// TIA Portal V17 export
// export: Created 2023-04-03T06:31:28.5466402Z, ExportSetting WithDefaults, DisplayName Totally Integrated Automation Portal, DisplayVersion V17 Update 4, DisplayName TIA Portal Openness, DisplayVersion V17 Update 4, DisplayName TIA Portal Version Control Interface, DisplayVersion V17, DisplayName STEP 7 Professional, DisplayVersion V17 Update 4, DisplayName STEP 7 Safety, DisplayVersion V17, DisplayName WinCC Professional, DisplayVersion V17 Update 4
DATA_BLOCK "PCS_2"   // DB43
{ S7_Optimized_Access := 'TRUE' }
VERSION : 0.1
// stored: AutoNumber true, DBAccessibleFromOPCUA true, DBAccessibleFromWebserver true, IsOnlyStoredInLoadMemory false, IsRetainMemResEnabled false, IsWriteProtectedInAS false, MemoryReserve 100
   VAR RETAIN
      TCONR_slow { S7_SetPoint := 'True'} : TCON_IP_v4;
   END_VAR
   VAR
      arrDataR_slow : Array[1..125] of Word;
      xREQR_slow : Bool;
      iCountDoneR_slow : Int := 1;
      iCountReadR_slow : Int := 1;
      MBmodeR_slow : USInt;
      MBdataAddrR_slow : UDInt;
      MBdataLenR_slow : UInt;
   END_VAR
   VAR RETAIN
      TCONR_fast { S7_SetPoint := 'True'} : TCON_IP_v4;
   END_VAR
   VAR
      arrDataR_fast : Array[1..125] of Word;
      xREQR_fast : Bool;
      iCountDoneR_fast : Int := 1;
      iCountReadR_fast : Int := 1;
      MBmodeR_fast : USInt;
      MBdataAddrR_fast : UDInt;
      MBdataLenR_fast : UInt;
   END_VAR
   VAR RETAIN
      TCONW_slow { S7_SetPoint := 'True'} : TCON_IP_v4;
   END_VAR
   VAR
      arrDataW_slow : Array[1..125] of Word;
      xREQW_slow : Bool;
      iCountDoneW_slow : Int := 1;
      iCountReadW_slow : Int := 1;
      MBmodeW_slow : USInt;
      MBdataAddrW_slow : UDInt;
      MBdataLenW_slow : UInt;
   END_VAR
   VAR RETAIN
      TCONW_fast { S7_SetPoint := 'True'} : TCON_IP_v4;
   END_VAR
   VAR
      arrDataW_fast : Array[1..125] of Word;
      xREQW_fast : Bool;
      iCountDoneW_fast : Int := 1;
      iCountReadW_fast : Int := 1;
      MBmodeW_fast : USInt;
      MBdataAddrW_fast : UDInt;
      MBdataLenW_fast : UInt;
      "____FINE SEGNALI CLIENT_____" : UInt;
      R { S7_SetPoint := 'True'} : "R_PE";
      RW { S7_SetPoint := 'True'} : "RW_PE";
      W { S7_SetPoint := 'True'} : "W_PE";
      arrStatus { S7_SetPoint := 'True'} : Array[0..17] of Bool;
      xDCbusAvl : Bool;
      xLVRT : Bool;
      xOVRT : Bool;
      xCommFltSt : Bool;
      xFltSt : Bool;
      xWarnSt : Bool;
      xModFltBus1St : Bool;
      xModFltBus2St : Bool;
      xMod1FltSt : Bool;
      xMod2FltSt : Bool;
      xMod3FltSt : Bool;
      xMod4FltSt : Bool;
      xMod5FltSt : Bool;
      xMod6FltSt : Bool;
      xMod1WarnSt : Bool;
      xMod2WarnSt : Bool;
      xMod3WarnSt : Bool;
      xMod4WarnSt : Bool;
      xMod5WarnSt : Bool;
      xMod6WarnSt : Bool;
      rMod1MaxTemp : Real;
      rMod2MaxTemp : Real;
      rMod3MaxTemp : Real;
      rMod4MaxTemp : Real;
      rMod5MaxTemp : Real;
      rMod6MaxTemp : Real;
      rPacBus1Meas : Real;
      rPacBus2Meas : Real;
      rQacBus1Meas : Real;
      rQacBus2Meas : Real;
      rLVacMeas : Real;
      rMVacMeas : Real;
      rIacTotMeas : Real;
      iCodeFlt : Int;
      iCodeWarn : Int;
      iModFlt : Int;
      iModWarn : Int;
      iLVac_Treshold : Int := 600;
      "____INVERTER FAULTS____" : Int;
      wInvFlt1 : Word;
      wInvFlt2 : Word;
      wInvFlt3 : Word;
      wInvFlt4 : Word;
      wInvFlt5 : Word;
      wInvFlt6 : Word;
      wInvFlt7 : Word;
      wInvWarn1 : Word;
      wInvWarn2 : Word;
      wInvWarn3 : Word;
      wInvWarn4 : Word;
      wInvWarn5 : Word;
      wInvWarn6 : Word;
      wMod1Flt1 : Word;
      wMod1Flt2 : Word;
      wMod1Flt3 : Word;
      wMod1Flt4 : Word;
      wMod2Flt1 : Word;
      wMod2Flt2 : Word;
      wMod2Flt3 : Word;
      wMod2Flt4 : Word;
      wMod3Flt1 : Word;
      wMod3Flt2 : Word;
      wMod3Flt3 : Word;
      wMod3Flt4 : Word;
      wMod4Flt1 : Word;
      wMod4Flt2 : Word;
      wMod4Flt3 : Word;
      wMod4Flt4 : Word;
      wMod5Flt1 : Word;
      wMod5Flt2 : Word;
      wMod5Flt3 : Word;
      wMod5Flt4 : Word;
      wMod6Flt1 : Word;
      wMod6Flt2 : Word;
      wMod6Flt3 : Word;
      wMod6Flt4 : Word;
      wMod1Warn1 : Word;
      wMod1Warn2 : Word;
      wMod1Warn3 : Word;
      wMod1Warn4 : Word;
      wMod2Warn1 : Word;
      wMod2Warn2 : Word;
      wMod2Warn3 : Word;
      wMod2Warn4 : Word;
      wMod3Warn1 : Word;
      wMod3Warn2 : Word;
      wMod3Warn3 : Word;
      wMod3Warn4 : Word;
      wMod4Warn1 : Word;
      wMod4Warn2 : Word;
      wMod4Warn3 : Word;
      wMod4Warn4 : Word;
      wMod5Warn1 : Word;
      wMod5Warn2 : Word;
      wMod5Warn3 : Word;
      wMod5Warn4 : Word;
      wMod6Warn1 : Word;
      wMod6Warn2 : Word;
      wMod6Warn3 : Word;
      wMod6Warn4 : Word;
      "_____TEST SIGNALS______" : Bool;
      xTestCmd : Bool;
      xTestRunCmd : Bool;
      xTestStopCmd : Bool;
      xTestResetCmd : Bool;
      xTestEnableCmd : Bool;
      xTestEmeCmd : Bool;
      "____SIGNAL EDGE______" : Bool;
      PSE : Struct
         x1 : Bool;
         x2 : Bool;
         x3 : Bool;
         x4 : Bool;
         x5 : Bool;
         x6 : Bool;
         x7 : Bool;
         x8 : Bool;
         x9 : Bool;
         x10 : Bool;
      END_STRUCT;
      NSE : Struct
         x1 : Bool;
         x2 : Bool;
         x3 : Bool;
         x4 : Bool;
         x5 : Bool;
         x6 : Bool;
         x7 : Bool;
         x8 : Bool;
         x9 : Bool;
         x10 : Bool;
      END_STRUCT;
   END_VAR
BEGIN
   TCONR_slow.RemoteAddress.ADDR[1] := 192;
   TCONR_slow.RemoteAddress.ADDR[2] := 168;
   TCONR_slow.RemoteAddress.ADDR[3] := 150;
   TCONR_slow.RemoteAddress.ADDR[4] := 44;
   TCONR_fast.RemoteAddress.ADDR[1] := 192;
   TCONR_fast.RemoteAddress.ADDR[2] := 168;
   TCONR_fast.RemoteAddress.ADDR[3] := 150;
   TCONR_fast.RemoteAddress.ADDR[4] := 44;
   // TCONW_slow.InterfaceId : HW_slow-identifier of IE-interface submodule
   TCONW_slow.RemoteAddress.ADDR[1] := 192;
   TCONW_slow.RemoteAddress.ADDR[2] := 168;
   TCONW_slow.RemoteAddress.ADDR[3] := 150;
   TCONW_slow.RemoteAddress.ADDR[4] := 44;
   TCONW_fast.RemoteAddress.ADDR[1] := 192;
   TCONW_fast.RemoteAddress.ADDR[2] := 168;
   TCONW_fast.RemoteAddress.ADDR[3] := 150;
   TCONW_fast.RemoteAddress.ADDR[4] := 44;
   // R.iCurrentStatus : Register 41004| 0:power up; 1:init; 2:off; 3:stanby DC; 4:precharge DC; 5:softcharge DC; 6:ready DC; 7:standby DC; 8:blackstart; 9:ready; 10:wait; 11:pre on; 12:on; 13:stop; 14:ready AC; 15:diagnostic AC; 16:discharge; 17:fault;
   // arrStatus[0] : power up
   // arrStatus[1] : init
   // arrStatus[2] : off
   // arrStatus[3] : standby DC
   // arrStatus[4] : precharge DC
   // arrStatus[5] : softcharge DC
   // arrStatus[6] : ready DC
   // arrStatus[7] : standby AC
   // arrStatus[8] : blackstart
   // arrStatus[9] : ready
   // arrStatus[10] : wait
   // arrStatus[11] : pre on
   // arrStatus[12] : on
   // arrStatus[13] : stop
   // arrStatus[14] : ready AC
   // arrStatus[15] : diagnostic AC
   // arrStatus[16] : discharge
   // arrStatus[17] : fault
END_DATA_BLOCK
